// TwinCAT 3 PLC project Aufgabenserie2
// ProgramVersion: 3.1.4022.3
// libraries:
//   Tc2_Standard, * (Beckhoff Automation GmbH)
//   Tc2_System, * (Beckhoff Automation GmbH)
//   Tc3_Module, * (Beckhoff Automation GmbH)
// project tree:
//   / GlobalTextList.TcGTLO, PlcTask.TcTTO, Visualisierungsmanager.TcVMO (not stored)
//   GVLs/ GVL.TcGVL
//   POUs/ AdditionFunction.TcPOU, DivisionFunction.TcPOU, DoSomeMath.TcPOU, MAIN.TcPOU, MultiplicationFunction.TcPOU, averageCalculator.TcPOU, Forgetting_Factor.TcPOU, shiftleft.TcPOU, SinusFunction.TcPOU (not stored), SquareSignal.TcPOU (not stored), SubtractionFunction.TcPOU
//   VISUs/ Visualization.TcVIS
// real-time tasks:
//   TASK PlcTask: cycle T#10ms, priority 20, ADS port 350
// I/O:
//   DEVICE Gerät 1 (EtherCAT) (disabled), AmsNetId 10.155.122.125.2.1
//     Klemme 1 (EK1200) [EK1200-5000 EtherCAT Netzteil (2A E-Bus)]
//       Klemme 2 (EL1004) [EL1004 4K. Dig. Eingang 24V, 3ms]
//       Klemme 3 (EL2004) [EL2004 4K. Dig. Ausgang 24V, 0.5A]
//       Klemme 4 (EL3004) [EL3004 4K.Ana. Eingang  +/-10V]
//       Klemme 5 (EL4034) [EL4034 4K. Ana. Ausgang +/-10V, 12bit]
//       Klemme 6 (EK1110) [EK1110 EtherCAT-Verlängerung]
// variable links:
//   Aufgabenserie2/Aufgabenserie2 Instance <-> Device 1 (EtherCAT)/Term 1 (EK1200)/Term 4 (EL3004)
//     PlcTask Inputs/GVL.i_UltrasonicSensor <-> AI Standard Channel 1/UltraschallSensor
//   Aufgabenserie2/Aufgabenserie2 Instance <-> Device 1 (EtherCAT)/Term 1 (EK1200)/Term 5 (EL4034)
//     PlcTask Outputs/GVL.i_voltageUltrasonicSensor <-> AO Outputs Channel 1/AnalogVoltage

CONFIGURATION Aufgabenserie2
    RESOURCE PLC ON TwinCAT3
        TASK PlcTask(INTERVAL := T#10ms, PRIORITY := 20);
        PROGRAM MAIN WITH PlcTask : MAIN;
    END_RESOURCE
END_CONFIGURATION

// ---- GVLs/GVL.TcGVL
{attribute 'qualified_only'}
VAR_GLOBAL
	i_UltrasonicSensor AT %I* : INT;
	i_voltageUltrasonicSensor AT %Q* : INT;
	r_bufferUltraschall : ARRAY [1..100] OF REAL;
END_VAR

// ---- POUs/MAIN.TcPOU
PROGRAM MAIN
VAR
	i_Result : REAL;
	i_OperandA : REAL;
	i_OperandB : REAL;
	r_FunctionSin : REAL;
	r_FunctionRec : REAL;
	u_Zykluszeit : UDINT := 0;
	r_MeanValSin : REAL;
	r_MeanValRec : REAL;
	r_AmplitudeSin : REAL := 1.3;
	r_OffsetSin : REAL := 0.4;
	r_MaxValueRec : REAL:= 2;
	r_MinValueRec : REAL := -2.1;
	r_KreisfrequenzSin : REAL := 10;
	r_KreisfrequenzRec : REAL := 23;
	r_ValuesSin : ARRAY[1..100] OF REAL;
    r_ValuesRec : ARRAY[1..100] OF REAL;
	r_FogettingFactor : REAL := 0.5;
	r_MeanValSinWithForget : REAL;	
	r_MeanValRecWithForget : REAL;
	func_forgetSin : Forgetting_Factor;
	func_forgetRec : Forgetting_Factor;
	
	sText : STRING := 'coucou';
	bButton : BOOL;
	rSlider : REAL;
END_VAR

i_Result := DivisionFunction(i_rValueA := 15.3 , i_rValueB :=5.1);
u_Zykluszeit := u_Zykluszeit +10;
r_FunctionSin := SinusFunction(r_Amplitude :=r_AmplitudeSin,r_Offset := r_OffsetSin, r_Kreisfrequenz := r_KreisfrequenzSin, r_Time := UDINT_TO_REAL(u_Zykluszeit)/1000);
r_FunctionRec := SquareSignal(r_MinValue := r_MinValueRec, r_MaxValue := r_MaxValueRec, r_Offset := 1,r_Kreisfrequenz:=r_KreisfrequenzRec, r_Time:= UDINT_TO_REAL(u_Zykluszeit)/1000);
GVL.i_voltageUltrasonicSensor := 32767-	GVL.i_UltrasonicSensor;
r_ValuesSin[100] := r_FunctionSin;
r_ValuesRec[100] := r_FunctionRec;
r_ValuesSin := shiftleft(r_ArrayInput := r_ValuesSin);
r_ValuesRec := shiftleft(r_ArrayInput := r_ValuesRec);
r_MeanValSin := averageCalculator(r_ValueInput := r_ValuesSin);
r_MeanValRec := averageCalculator(r_ValueInput := r_ValuesRec);

func_forgetSin();
func_forgetSin.r_forgetFactor := r_FogettingFactor;
func_forgetSin.r_inputValue := r_FunctionSin;
r_MeanValSinWithForget := func_forgetSin.r_meanValueForget_k;

func_forgetRec();
func_forgetRec.r_forgetFactor := r_FogettingFactor;
func_forgetRec.r_inputValue := r_FunctionRec;
r_MeanValRecWithForget := func_forgetRec.r_meanValueForget_k;

END_PROGRAM

// ---- POUs/Forgetting_Factor.TcPOU
FUNCTION_BLOCK Forgetting_Factor
VAR_INPUT
	r_forgetFactor : REAL;
	r_inputValue : REAL;
END_VAR
VAR_OUTPUT
	r_meanValueForget_k : REAL;
END_VAR
VAR
	r_meanValueForget_k1 : REAL;
END_VAR

r_meanValueForget_k := r_meanValueForget_k1*r_forgetFactor + (1-r_forgetFactor)*r_inputValue;
r_meanValueForget_k1 := r_meanValueForget_k;

END_FUNCTION_BLOCK

// ---- POUs/DivisionFunction.TcPOU
FUNCTION DivisionFunction : REAL
VAR_INPUT
	i_rValueA : REAL;
	i_rValueB : REAL;
END_VAR
VAR
END_VAR

IF	i_rValueB <> 0 THEN
DivisionFunction := i_rValueA / i_rValueB;
ELSE
	DivisionFunction := 0;
END_IF

END_FUNCTION

// ---- POUs/shiftleft.TcPOU
FUNCTION shiftleft : ARRAY[1..100] OF REAL;
VAR_INPUT
	r_ArrayInput : ARRAY[1..100] OF REAL;
END_VAR
VAR
	r_ArrayOutput : ARRAY[1..100] OF REAL;
	i_index : INT;
END_VAR

FOR i_index := 2  TO 100 BY 1 DO
	r_ArrayOutput[i_index-1] := r_ArrayInput[i_index];
END_FOR
shiftleft := r_ArrayOutput;

END_FUNCTION

// ---- POUs/averageCalculator.TcPOU
FUNCTION averageCalculator : REAL
VAR_INPUT
	r_ValueInput : ARRAY[1..100] OF REAL;
END_VAR
VAR
	i_Index : INT;
	r_MeanValue : REAL := 0;
END_VAR

FOR i_Index := 1 TO 100 BY 1 DO
	r_MeanValue := r_MeanValue + r_ValueInput[i_Index];
END_FOR

averageCalculator := r_MeanValue/100;

END_FUNCTION

// ---- POUs/AdditionFunction.TcPOU
FUNCTION AdditionFunction : REAL
VAR_INPUT
	i_rValueA : REAL;
	i_rValueB : REAL;
END_VAR
VAR
END_VAR

AdditionFunction := i_rValueA + i_rValueB;

END_FUNCTION

// ---- POUs/DoSomeMath.TcPOU
PROGRAM DoSomeMath
VAR_INPUT
	i_rInputA: REAL;
	i_rInputB: REAL;
END_VAR
VAR
END_VAR

END_PROGRAM

// ---- POUs/MultiplicationFunction.TcPOU
FUNCTION MultiplicationFunction : REAL
VAR_INPUT
	i_rValueA : REAL;
	i_rValueB : REAL;
END_VAR
VAR
END_VAR

MultiplicationFunction := i_rValueA * i_rValueB;

END_FUNCTION

// ---- POUs/SubtractionFunction.TcPOU
FUNCTION SubtractionFunction : REAL
VAR_INPUT
	i_rValueA : REAL;
	i_rValueB : REAL;
VAR
END_VAR

SubtractionFunction := i_rValueA - i_rValueB;

END_FUNCTION

// ---- GlobalTextList.TcGTLO
TEXTLIST GlobalTextList
  73 = '%s'
  976 = 'Amplitude Sin'
  452 = 'Fogetting Factor'
  523 = 'Max Rectangle'
  831 = 'Min Rectangle'
  339 = 'Offset Sin'
  643 = 'rad/s Rec'
  230 = 'rad/s Sin'
END_TEXTLIST

// ---- VISUs/Visualization.TcVIS
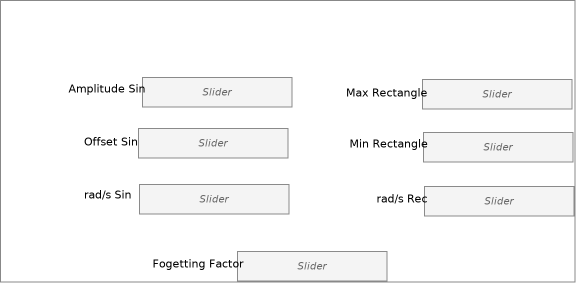
VISUALIZATION Visualization  // 576x283
    Slider (142,77 150x30), variable: MAIN.r_AmplitudeSin, scale 0..50
    Label (32,74 150x30), "Amplitude Sin"
    Slider (422,79 150x30), variable: MAIN.r_MaxValueRec, scale 0..50
    Label (312,78 150x30), "Max Rectangle"
    Slider (423,132 150x30), variable: MAIN.r_MinValueRec, scale -50..0
    Label (314,129 150x30), "Min Rectangle"
    Slider (139,184 150x30), variable: MAIN.r_KreisfrequenzSin, scale 0..100
    Label (33,180 150x30), "rad/s Sin"
    Slider (424,186 150x30), variable: MAIN.r_KreisfrequenzRec, scale 0..100
    Label (327,184 150x30), "rad/s Rec"
    Slider (138,128 150x30), variable: MAIN.r_OffsetSin, scale -20..20
    Label (36,127 150x30), "Offset Sin"
    Slider (237,251 150x30), variable: MAIN.r_FogettingFactor, scale 0..0.999
    Label (123,249 150x30), "Fogetting Factor"
END_VISUALIZATION
